FUNCTION_BLOCK FB_System_BSp_797
VAR_INPUT
	Freigabe_auto			: BOOL;
	Freigabe_Deakt_auto		: BOOL;
	Betrieb_Anford_auto		: BOOL;

	Regelung_Modus_auto		: SINT;
	Regelung_Sollw_auto		: REAL;

	Temp_Netz_WW			: REAL;
END_VAR
VAR_OUTPUT
	{attribute 'OPC.UA.DA' := '1'}Steuerung				: ST_System_BSp_Steuerung;		
	{attribute 'OPC.UA.DA' := '1'}Stellwert					: ST_System_BSp_Stellwert;	
	{attribute 'OPC.UA.DA' := '1'}Zustand					: ST_System_BSp_Zustand;	
	{attribute 'OPC.UA.DA' := '1'}Parameter				: ST_System_BSp_Parameter;		
END_VAR
VAR
	Stellventil_205			: FB_SV;
	Pumpe_205				: FB_PU;
	Pumpe_720				: FB_PU_Schuetz;
	Betonspeicher_797		: FB_BSp;

	Zustandscheck			: FB_System_BSp_797_Zustandscheck;
	Logik					: FB_System_BSp_Logik;
	Ablaufsteuerung			: FB_System_BSp_Ablaufsteuerung;
	Sollwertscheck			: FB_System_BSp_Sollwertscheck;
	Regelung				: FB_System_BSp_Regelung;
	Stellwertscheck			: FB_System_BSp_Stellwertscheck;
END_VAR
VAR // added by the converter: edge detectors and wires of the graphical bodies
    _w1, _w2 : ANY;
END_VAR

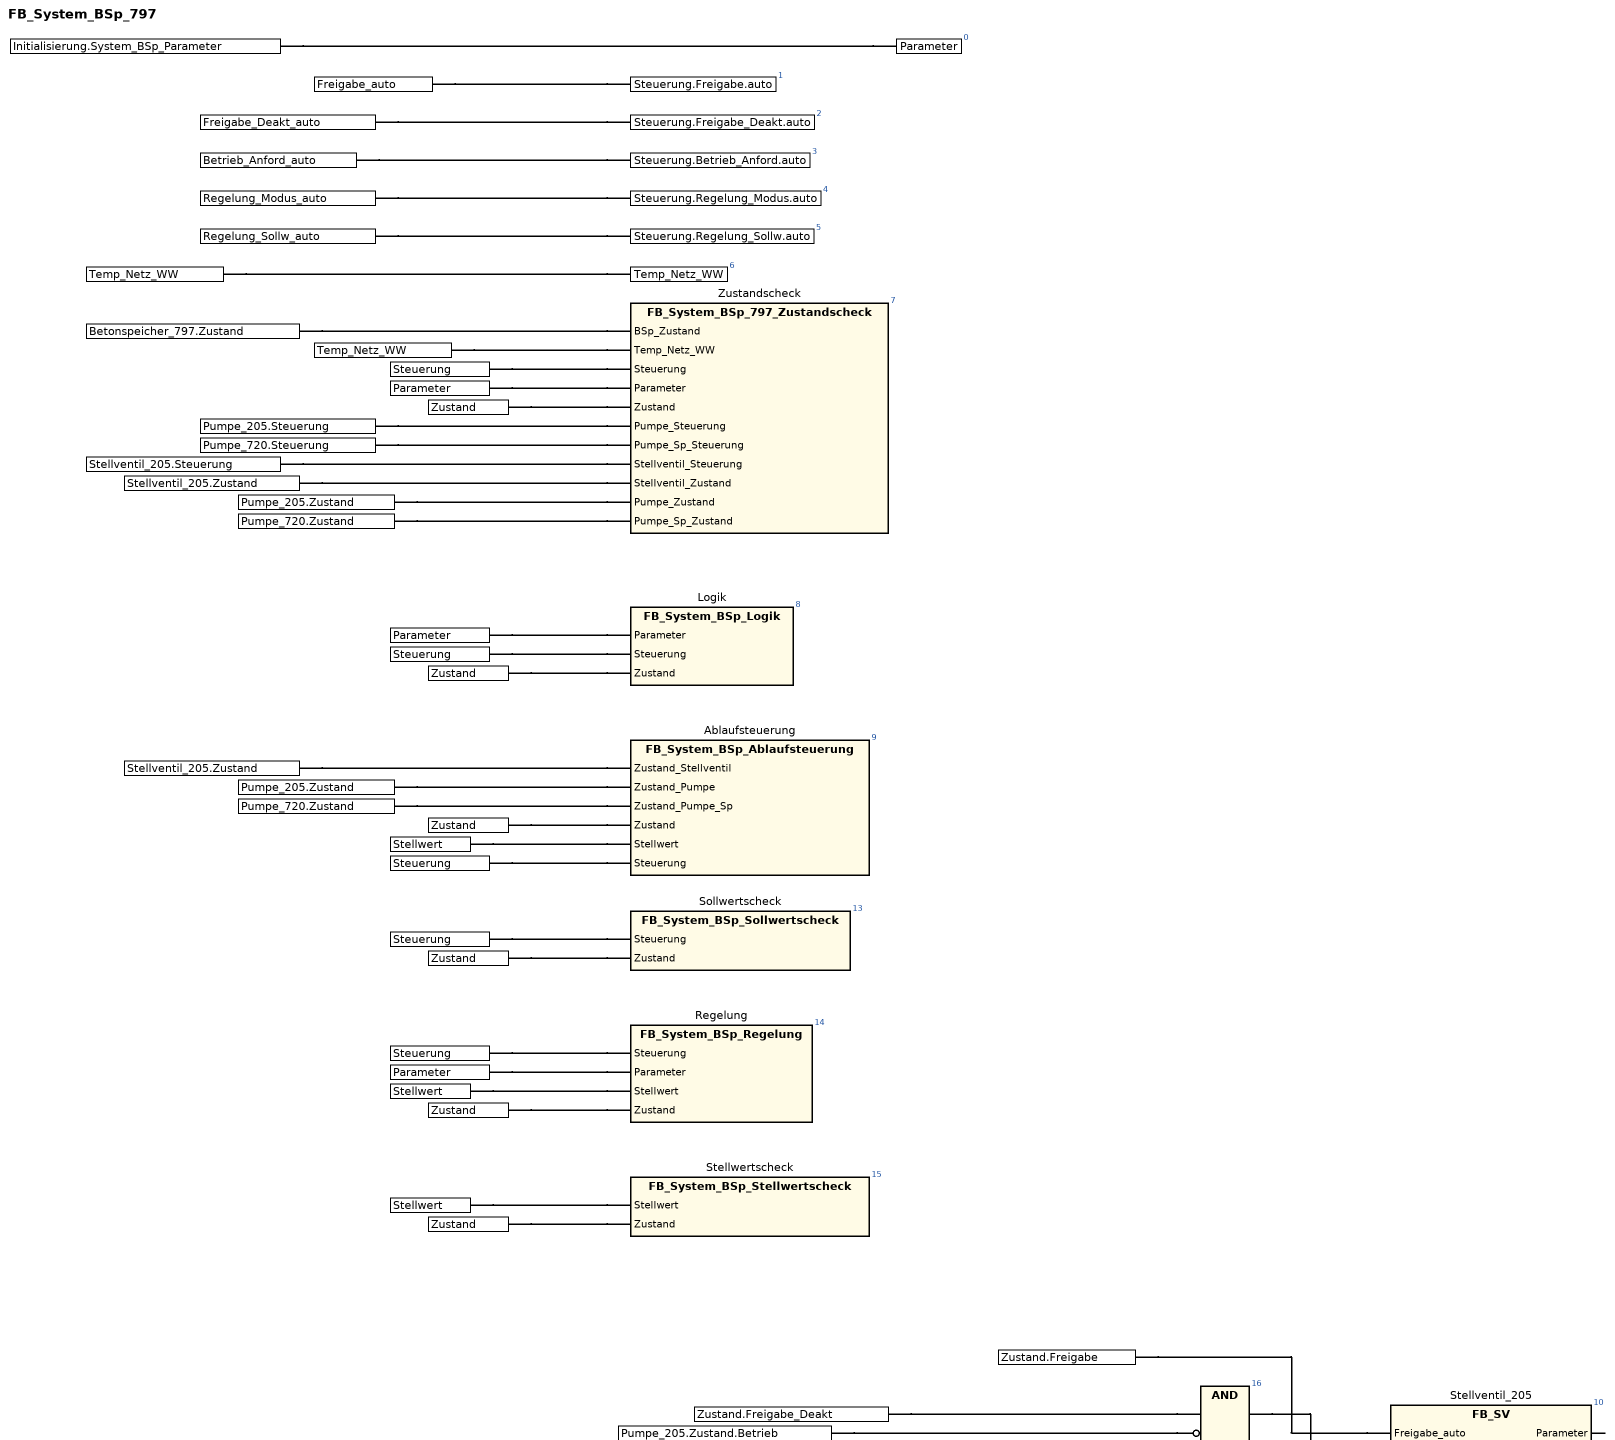
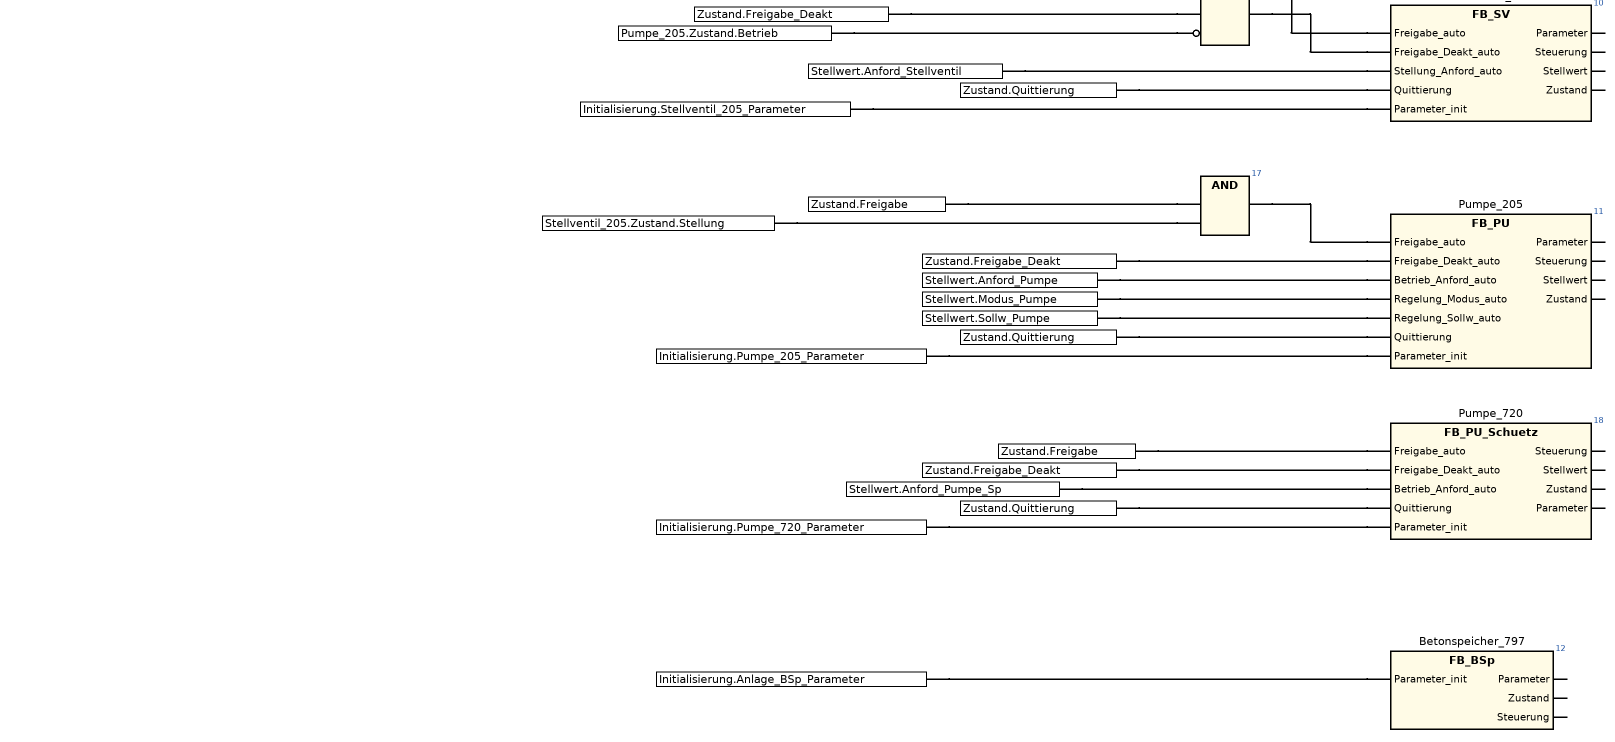
Parameter := Initialisierung.System_BSp_Parameter;
Steuerung.Freigabe.auto := Freigabe_auto;
Steuerung.Freigabe_Deakt.auto := Freigabe_Deakt_auto;
Steuerung.Betrieb_Anford.auto := Betrieb_Anford_auto;
Steuerung.Regelung_Modus.auto := Regelung_Modus_auto;
Steuerung.Regelung_Sollw.auto := Regelung_Sollw_auto;
Temp_Netz_WW := Temp_Netz_WW;
Zustandscheck(
    BSp_Zustand := Betonspeicher_797.Zustand,
    Temp_Netz_WW := Temp_Netz_WW,
    Steuerung := Steuerung,
    Parameter := Parameter,
    Zustand := Zustand,
    Pumpe_Steuerung := Pumpe_205.Steuerung,
    Pumpe_Sp_Steuerung := Pumpe_720.Steuerung,
    Stellventil_Steuerung := Stellventil_205.Steuerung,
    Stellventil_Zustand := Stellventil_205.Zustand,
    Pumpe_Zustand := Pumpe_205.Zustand,
    Pumpe_Sp_Zustand := Pumpe_720.Zustand); // FB_System_BSp_797_Zustandscheck
Logik(Parameter := Parameter, Steuerung := Steuerung, Zustand := Zustand); // FB_System_BSp_Logik
Ablaufsteuerung(
    Zustand_Stellventil := Stellventil_205.Zustand,
    Zustand_Pumpe := Pumpe_205.Zustand,
    Zustand_Pumpe_Sp := Pumpe_720.Zustand,
    Zustand := Zustand,
    Stellwert := Stellwert,
    Steuerung := Steuerung); // FB_System_BSp_Ablaufsteuerung
Stellventil_205(
    Freigabe_auto := Zustand.Freigabe,
    Freigabe_Deakt_auto := _w1,
    Stellung_Anford_auto := Stellwert.Anford_Stellventil,
    Quittierung := Zustand.Quittierung,
    Parameter_init := Initialisierung.Stellventil_205_Parameter); // FB_SV
Pumpe_205(
    Freigabe_auto := _w2,
    Freigabe_Deakt_auto := Zustand.Freigabe_Deakt,
    Betrieb_Anford_auto := Stellwert.Anford_Pumpe,
    Regelung_Modus_auto := Stellwert.Modus_Pumpe,
    Regelung_Sollw_auto := Stellwert.Sollw_Pumpe,
    Quittierung := Zustand.Quittierung,
    Parameter_init := Initialisierung.Pumpe_205_Parameter); // FB_PU
Betonspeicher_797(Parameter_init := Initialisierung.Anlage_BSp_Parameter); // FB_BSp
Sollwertscheck(Steuerung := Steuerung, Zustand := Zustand); // FB_System_BSp_Sollwertscheck
Regelung(Steuerung := Steuerung, Parameter := Parameter, Stellwert := Stellwert, Zustand := Zustand); // FB_System_BSp_Regelung
Stellwertscheck(Stellwert := Stellwert, Zustand := Zustand); // FB_System_BSp_Stellwertscheck
_w1 := Zustand.Freigabe_Deakt AND NOT Pumpe_205.Zustand.Betrieb;
_w2 := Zustand.Freigabe AND Stellventil_205.Zustand.Stellung;
Pumpe_720(
    Freigabe_auto := Zustand.Freigabe,
    Freigabe_Deakt_auto := Zustand.Freigabe_Deakt,
    Betrieb_Anford_auto := Stellwert.Anford_Pumpe_Sp,
    Quittierung := Zustand.Quittierung,
    Parameter_init := Initialisierung.Pumpe_720_Parameter); // FB_PU_Schuetz

END_FUNCTION_BLOCK

(* stored: Version 1.1.0.1, ProductVersion 3.1.4024.9
   POU FB_System_BSp_797: Id {17e203a9-91d2-4997-b2fa-3d75abb9c0b9}, SpecialFunc None *)
